(* Logix 5000 project; controller Sucrose_Main Emulate 5570 rev 20.12; software revision 20.01; part 28 of 30 *)
(* tags used below, declared in another part *)
   AI_E23_0 : REAL[8];   // Analog Input EN2T_FLX 192.168.1.23
   AI_E23_1 : REAL[8];   // Analog Input EN2T_FLX 192.168.1.23
   Alarm_ACK_Master_Timer : TIMER;
   DI_E23_3 : ALIAS FOR FLX_E23:3:I;   // Discrete Input EN2T_FLX 192.168.1.23
   DO_E24_3 : ALIAS FOR FLX_E24:3:O;   // Discrete Output EN2T_FLX 192.168.1.24
   FV230102_AOI : QSI_Flow_Valve;   // FV-23-01-02 SUCROSE TANK #1 INLET/SPRAYBALL VALVE
   FV230104_AOI : QSI_Flow_Valve;   // FV-23-01-04-O SUCROSE RETURN TO SUCROSE TANK #1 VALVE OPEN
   FV230204_AOI : QSI_Flow_Valve;   // FV-23-02-04-O SUCROSE RETURN TO SUCROSE TANK #2 VALVE OPEN
   FV230222_AOI : QSI_Flow_Valve;   // FV-23-02-22-O SUCROSE TANK #2 TO TRANSFER PUMP #2 MIX PROOF VALVE OPEN
   FV230304_AOI : QSI_Flow_Valve;   // FV-23-03-04-O SUCROSE RETURN TO SUCROSE TANK #3 VALVE OPEN
   FV230411_AOI : QSI_Flow_Valve;   // FV-23-04-11-O SUCROSE TANK #1 TO TRANSFER PUMP #1 MIX PROOF VALVE OPEN
   FV230412_AOI : QSI_Flow_Valve;   // FV-23-04-12-O SUCROSE TANK #2 TO TRANSFER PUMP #1 MIX PROOF VALVE OPEN
   FV230413_AOI : QSI_Flow_Valve;   // FV-23-04-13-O SUCROSE TANK #3 TO TRANSFER PUMP #1 MIX PROOF VALVE OPEN
   FV230421_AOI : QSI_Flow_Valve;   // FV-23-04-21-O SUCROSE TANK #1 TO TRANSFER PUMP #2 MIX PROOF VALVE OPEN
   FV230423_AOI : QSI_Flow_Valve;   // FV-23-04-23-O SUCROSE TANK #3 TO TRANSFER PUMP #2 MIX PROOF VALVE OPEN
   FV751101_AOI : QSI_Flow_Valve;   // FV-75-11-01 SUCROSE TANK #1 BLANKETING STEAM TRAP ISOLATION VALVE
   FV931101_AOI : QSI_Flow_Valve;   // FV-93-11-01 STERILE AIR FLT-93-11-01 SHUT OFF VALVE
   ONESHOTBITS : INT[10];
   Rung_Comment : BOOL;
   Sucrose_MM_Enable : BOOL;
   SucroseCIP_RINGMAIN_REMOTE : CIP_REMOTE;
   SucroseCIP_TK230101_REMOTE : CIP_REMOTE;
   SucroseCIP_TK230201_REMOTE : CIP_REMOTE;
   SucroseCIP_TK230301_REMOTE : CIP_REMOTE;
   SucroseDischarge : Area_Program;
   SucroseFiltration : Area_Program;
   SucroseTanks : Area_Program;
   TK_23_01_01_HEALOUT_TIME_REMAINING : DINT;
   TK_23_01_01_LOW_LEVEL : DINT;
   TK_23_01_01_NO_PRESS_ALARM : BOOL;
   TK_23_01_01_NO_TEMP_ALARM : BOOL;
   TK_23_02_01_HEALOUT_TIME_REMAINING : DINT;
   TK_23_02_01_LOW_LEVEL : DINT;
   TK_23_02_01_NO_PRESS_ALARM : BOOL;
   TK_23_02_01_NO_TEMP_ALARM : BOOL;
   TK_23_03_01_HEALOUT_TIME_REMAINING : DINT;
   TK_23_03_01_LOW_LEVEL : DINT;
   TK_23_03_01_NO_PRESS_ALARM : BOOL;
   TK_23_03_01_NO_TEMP_ALARM : BOOL;
(* TanksArea_AutoLogic, continued *)

ROUTINE Control_Logic   (* ladder *)
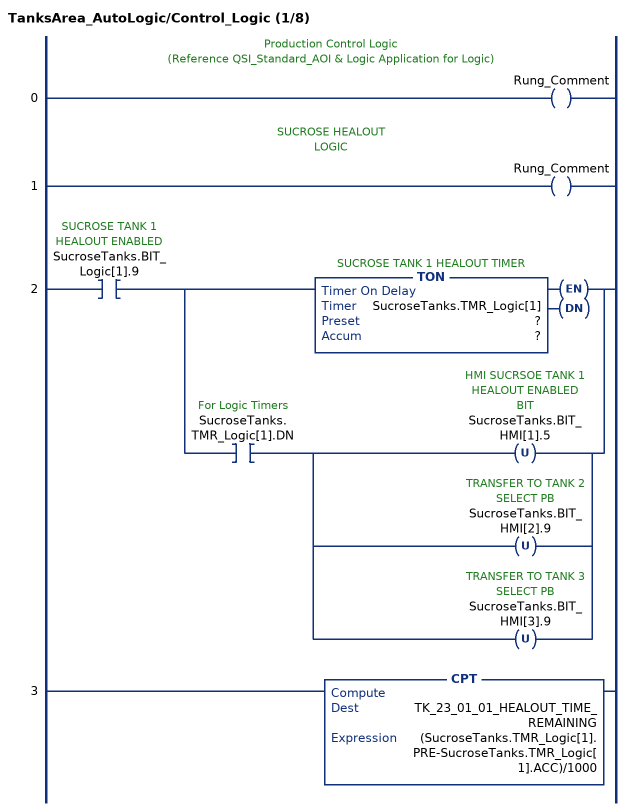
   // Production Control Logic
   // (Reference QSI_Standard_AOI & Logic Application for Logic)
   0: OTE(Rung_Comment);
   // SUCROSE HEALOUT
   // LOGIC
   1: OTE(Rung_Comment);
   2: XIC(SucroseTanks.BIT_Logic[1].9)[TON(SucroseTanks.TMR_Logic[1],?,?) ,XIC(SucroseTanks.TMR_Logic[1].DN) [OTU(SucroseTanks.BIT_HMI[1].5) ,OTU(SucroseTanks.BIT_HMI[2].9) ,OTU(SucroseTanks.BIT_HMI[3].9) ] ];
   3: CPT(TK_23_01_01_HEALOUT_TIME_REMAINING,(SucroseTanks.TMR_Logic[1].PRE-SucroseTanks.TMR_Logic[1].ACC)/1000);
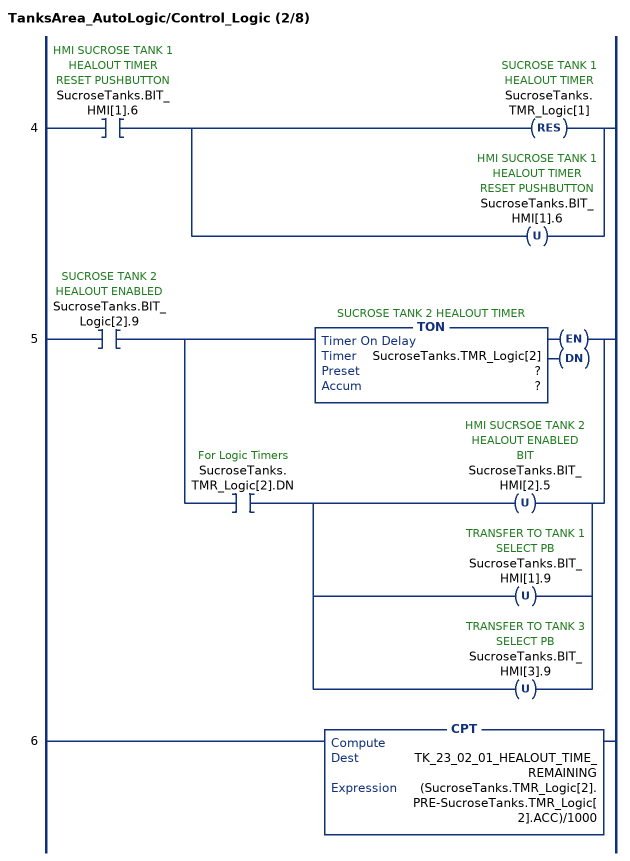
   4: XIC(SucroseTanks.BIT_HMI[1].6)[RES(SucroseTanks.TMR_Logic[1]) ,OTU(SucroseTanks.BIT_HMI[1].6) ];
   5: XIC(SucroseTanks.BIT_Logic[2].9)[TON(SucroseTanks.TMR_Logic[2],?,?) ,XIC(SucroseTanks.TMR_Logic[2].DN) [OTU(SucroseTanks.BIT_HMI[2].5) ,OTU(SucroseTanks.BIT_HMI[1].9) ,OTU(SucroseTanks.BIT_HMI[3].9) ] ];
   6: CPT(TK_23_02_01_HEALOUT_TIME_REMAINING,(SucroseTanks.TMR_Logic[2].PRE-SucroseTanks.TMR_Logic[2].ACC)/1000);
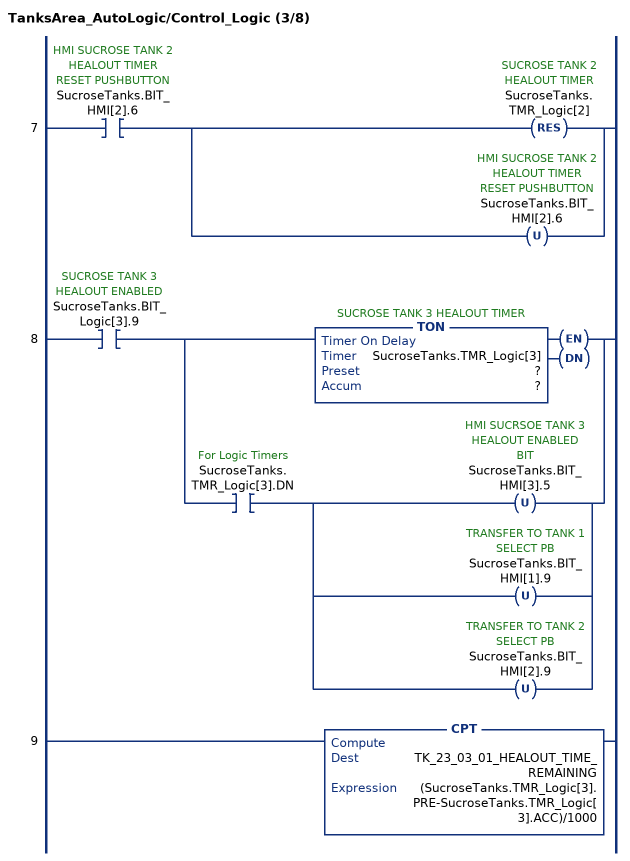
   7: XIC(SucroseTanks.BIT_HMI[2].6)[RES(SucroseTanks.TMR_Logic[2]) ,OTU(SucroseTanks.BIT_HMI[2].6) ];
   8: XIC(SucroseTanks.BIT_Logic[3].9)[TON(SucroseTanks.TMR_Logic[3],?,?) ,XIC(SucroseTanks.TMR_Logic[3].DN) [OTU(SucroseTanks.BIT_HMI[3].5) ,OTU(SucroseTanks.BIT_HMI[1].9) ,OTU(SucroseTanks.BIT_HMI[2].9) ] ];
   9: CPT(TK_23_03_01_HEALOUT_TIME_REMAINING,(SucroseTanks.TMR_Logic[3].PRE-SucroseTanks.TMR_Logic[3].ACC)/1000);
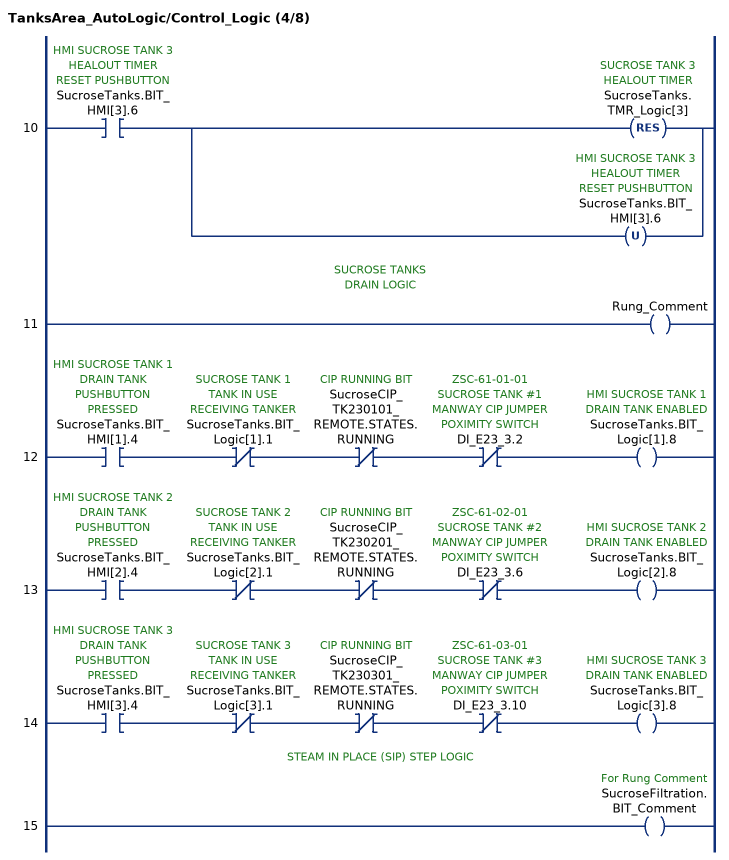
   10: XIC(SucroseTanks.BIT_HMI[3].6)[RES(SucroseTanks.TMR_Logic[3]) ,OTU(SucroseTanks.BIT_HMI[3].6) ];
   // SUCROSE TANKS
   // DRAIN LOGIC
   11: OTE(Rung_Comment);
   12: XIC(SucroseTanks.BIT_HMI[1].4)XIO(SucroseTanks.BIT_Logic[1].1)XIO(SucroseCIP_TK230101_REMOTE.STATES.RUNNING)XIO(DI_E23_3.2)OTE(SucroseTanks.BIT_Logic[1].8);
   13: XIC(SucroseTanks.BIT_HMI[2].4)XIO(SucroseTanks.BIT_Logic[2].1)XIO(SucroseCIP_TK230201_REMOTE.STATES.RUNNING)XIO(DI_E23_3.6)OTE(SucroseTanks.BIT_Logic[2].8);
   14: XIC(SucroseTanks.BIT_HMI[3].4)XIO(SucroseTanks.BIT_Logic[3].1)XIO(SucroseCIP_TK230301_REMOTE.STATES.RUNNING)XIO(DI_E23_3.10)OTE(SucroseTanks.BIT_Logic[3].8);
   // STEAM IN PLACE (SIP) STEP LOGIC
   15: OTE(SucroseFiltration.BIT_Comment);
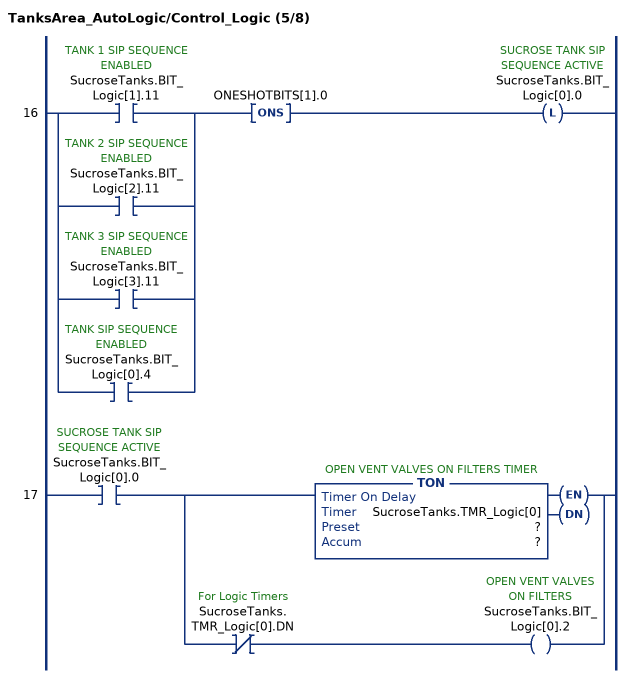
   16: [XIC(SucroseTanks.BIT_Logic[1].11) ,XIC(SucroseTanks.BIT_Logic[2].11) ,XIC(SucroseTanks.BIT_Logic[3].11) ,XIC(SucroseTanks.BIT_Logic[0].4) ]ONS(ONESHOTBITS[1].0)OTL(SucroseTanks.BIT_Logic[0].0);
   17: XIC(SucroseTanks.BIT_Logic[0].0)[TON(SucroseTanks.TMR_Logic[0],?,?) ,XIO(SucroseTanks.TMR_Logic[0].DN) OTE(SucroseTanks.BIT_Logic[0].2) ];
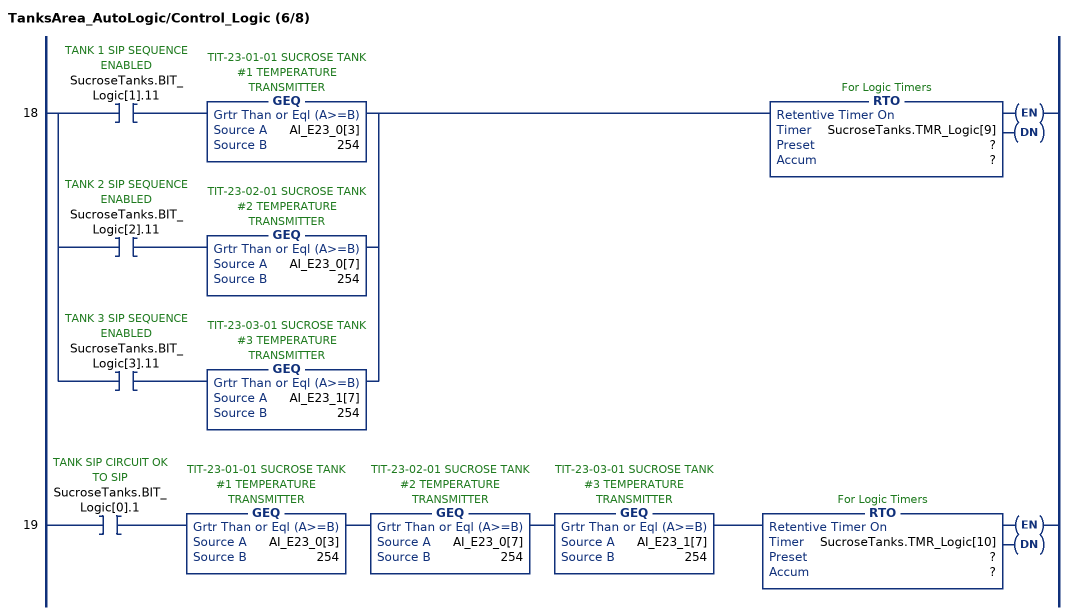
   18: [XIC(SucroseTanks.BIT_Logic[1].11) GEQ(AI_E23_0[3],254) ,XIC(SucroseTanks.BIT_Logic[2].11) GEQ(AI_E23_0[7],254) ,XIC(SucroseTanks.BIT_Logic[3].11) GEQ(AI_E23_1[7],254) ]RTO(SucroseTanks.TMR_Logic[9],?,?);
   19: XIC(SucroseTanks.BIT_Logic[0].1)GEQ(AI_E23_0[3],254)GEQ(AI_E23_0[7],254)GEQ(AI_E23_1[7],254)RTO(SucroseTanks.TMR_Logic[10],?,?);
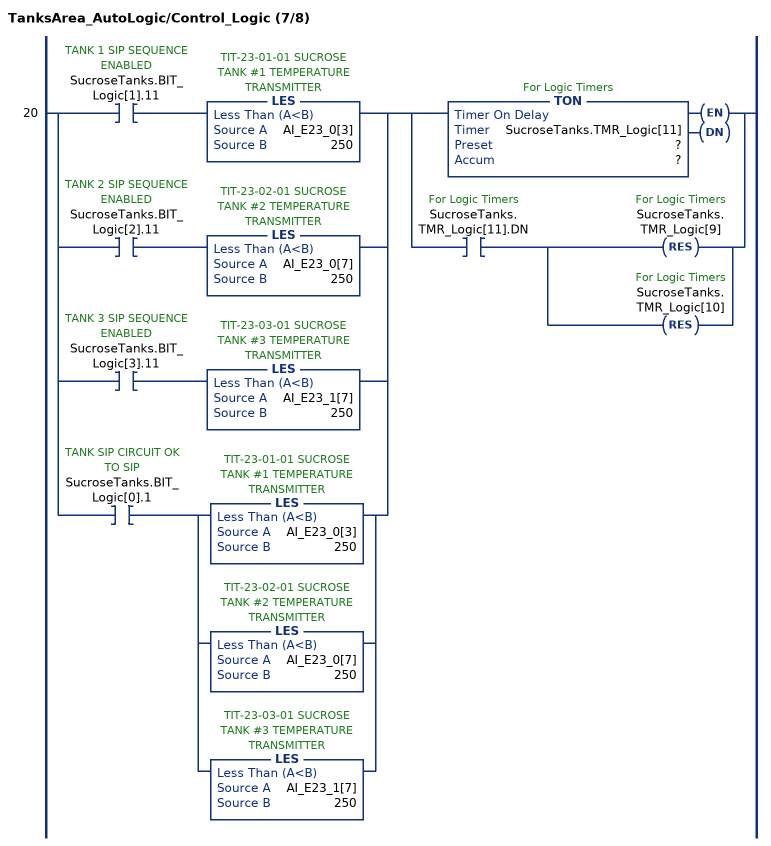
   20: [XIC(SucroseTanks.BIT_Logic[1].11) LES(AI_E23_0[3],250) ,XIC(SucroseTanks.BIT_Logic[2].11) LES(AI_E23_0[7],250) ,XIC(SucroseTanks.BIT_Logic[3].11) LES(AI_E23_1[7],250) ,XIC(SucroseTanks.BIT_Logic[0].1) [LES(AI_E23_0[3],250) ,LES(AI_E23_0[7],250) ,LES(AI_E23_1[7],250) ] ][TON(SucroseTanks.TMR_Logic[11],?,?) ,XIC(SucroseTanks.TMR_Logic[11].DN) [RES(SucroseTanks.TMR_Logic[9]) ,RES(SucroseTanks.TMR_Logic[10]) ] ];
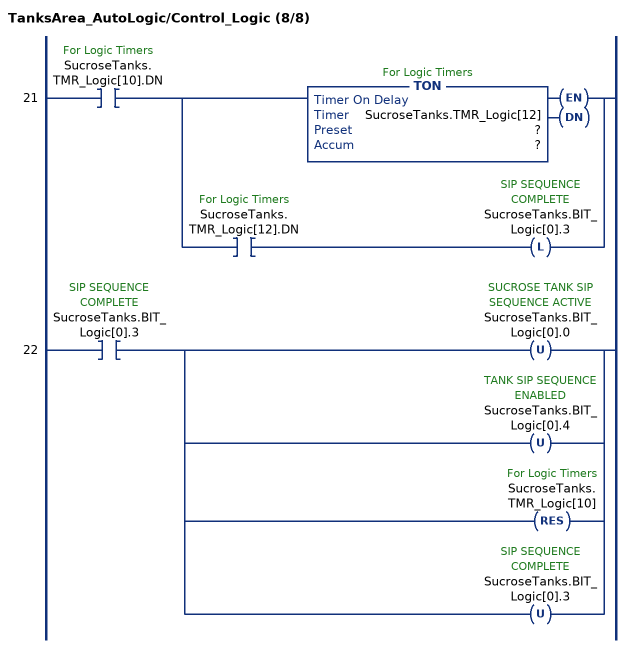
   21: XIC(SucroseTanks.TMR_Logic[10].DN)[TON(SucroseTanks.TMR_Logic[12],?,?) ,XIC(SucroseTanks.TMR_Logic[12].DN) OTL(SucroseTanks.BIT_Logic[0].3) ];
   22: XIC(SucroseTanks.BIT_Logic[0].3)[OTU(SucroseTanks.BIT_Logic[0].0) ,OTU(SucroseTanks.BIT_Logic[0].4) ,RES(SucroseTanks.TMR_Logic[10]) ,OTU(SucroseTanks.BIT_Logic[0].3) ];
END_ROUTINE

ROUTINE Enable_Logic   (* ladder *)
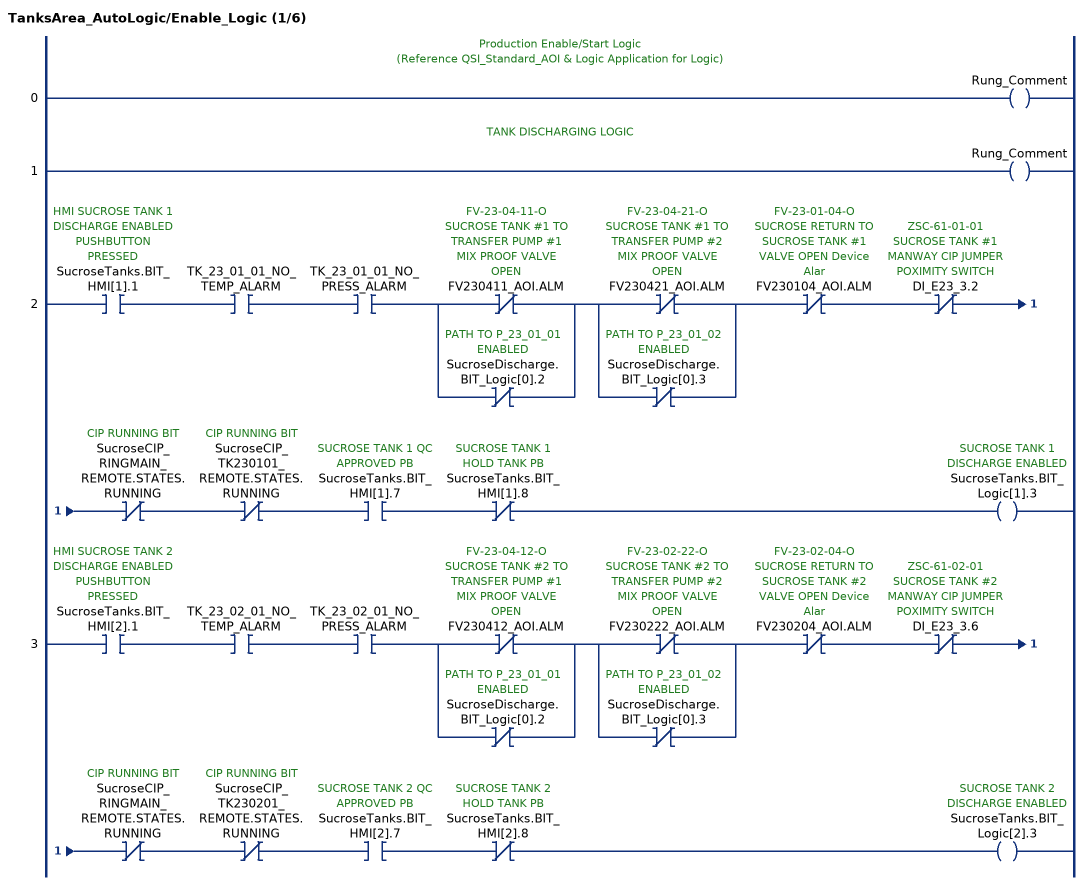
   // Production Enable/Start Logic
   // (Reference QSI_Standard_AOI & Logic Application for Logic)
   0: OTE(Rung_Comment);
   // TANK DISCHARGING LOGIC
   1: OTE(Rung_Comment);
   2: XIC(SucroseTanks.BIT_HMI[1].1)XIC(TK_23_01_01_NO_TEMP_ALARM)XIC(TK_23_01_01_NO_PRESS_ALARM)[XIO(FV230411_AOI.ALM) ,XIO(SucroseDischarge.BIT_Logic[0].2) ][XIO(FV230421_AOI.ALM) ,XIO(SucroseDischarge.BIT_Logic[0].3) ]XIO(FV230104_AOI.ALM)XIO(DI_E23_3.2)XIO(SucroseCIP_RINGMAIN_REMOTE.STATES.RUNNING)XIO(SucroseCIP_TK230101_REMOTE.STATES.RUNNING)XIC(SucroseTanks.BIT_HMI[1].7)XIO(SucroseTanks.BIT_HMI[1].8)OTE(SucroseTanks.BIT_Logic[1].3);
   3: XIC(SucroseTanks.BIT_HMI[2].1)XIC(TK_23_02_01_NO_TEMP_ALARM)XIC(TK_23_02_01_NO_PRESS_ALARM)[XIO(FV230412_AOI.ALM) ,XIO(SucroseDischarge.BIT_Logic[0].2) ][XIO(FV230222_AOI.ALM) ,XIO(SucroseDischarge.BIT_Logic[0].3) ]XIO(FV230204_AOI.ALM)XIO(DI_E23_3.6)XIO(SucroseCIP_RINGMAIN_REMOTE.STATES.RUNNING)XIO(SucroseCIP_TK230201_REMOTE.STATES.RUNNING)XIC(SucroseTanks.BIT_HMI[2].7)XIO(SucroseTanks.BIT_HMI[2].8)OTE(SucroseTanks.BIT_Logic[2].3);
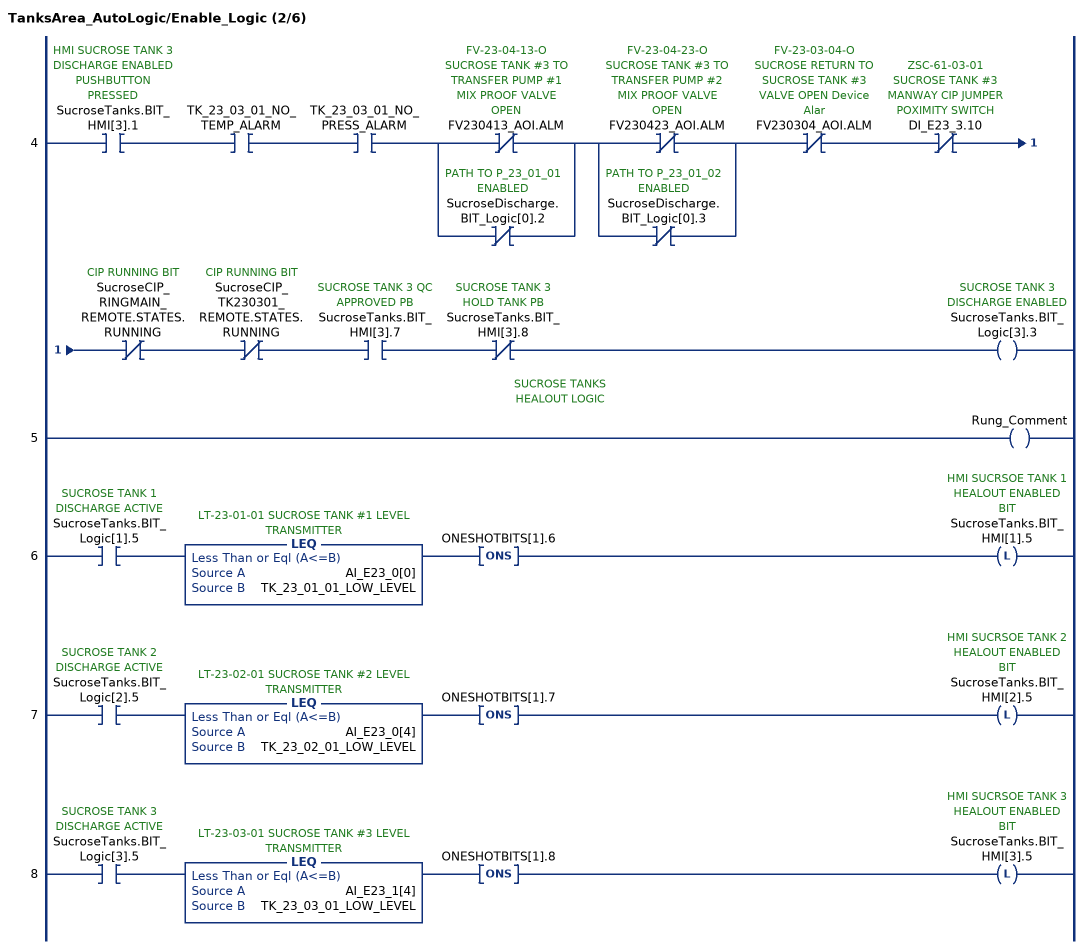
   4: XIC(SucroseTanks.BIT_HMI[3].1)XIC(TK_23_03_01_NO_TEMP_ALARM)XIC(TK_23_03_01_NO_PRESS_ALARM)[XIO(FV230413_AOI.ALM) ,XIO(SucroseDischarge.BIT_Logic[0].2) ][XIO(FV230423_AOI.ALM) ,XIO(SucroseDischarge.BIT_Logic[0].3) ]XIO(FV230304_AOI.ALM)XIO(DI_E23_3.10)XIO(SucroseCIP_RINGMAIN_REMOTE.STATES.RUNNING)XIO(SucroseCIP_TK230301_REMOTE.STATES.RUNNING)XIC(SucroseTanks.BIT_HMI[3].7)XIO(SucroseTanks.BIT_HMI[3].8)OTE(SucroseTanks.BIT_Logic[3].3);
   // SUCROSE TANKS
   // HEALOUT LOGIC
   5: OTE(Rung_Comment);
   6: XIC(SucroseTanks.BIT_Logic[1].5)LEQ(AI_E23_0[0],TK_23_01_01_LOW_LEVEL)ONS(ONESHOTBITS[1].6)OTL(SucroseTanks.BIT_HMI[1].5);
   7: XIC(SucroseTanks.BIT_Logic[2].5)LEQ(AI_E23_0[4],TK_23_02_01_LOW_LEVEL)ONS(ONESHOTBITS[1].7)OTL(SucroseTanks.BIT_HMI[2].5);
   8: XIC(SucroseTanks.BIT_Logic[3].5)LEQ(AI_E23_1[4],TK_23_03_01_LOW_LEVEL)ONS(ONESHOTBITS[1].8)OTL(SucroseTanks.BIT_HMI[3].5);
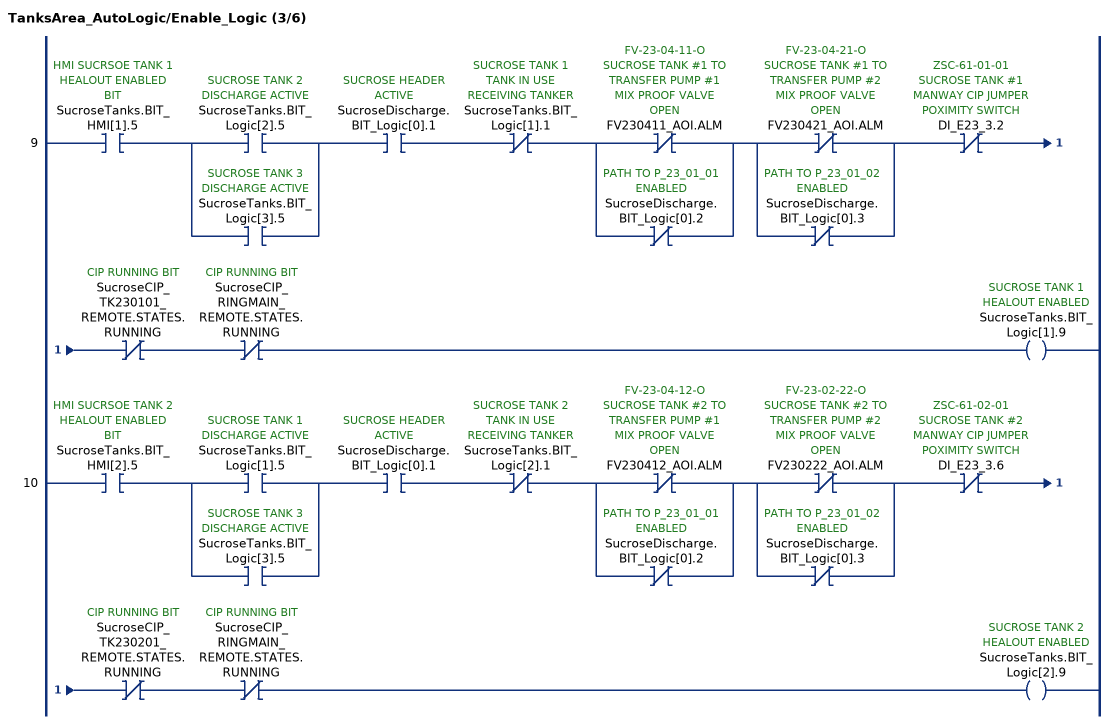
   9: XIC(SucroseTanks.BIT_HMI[1].5)[XIC(SucroseTanks.BIT_Logic[2].5) ,XIC(SucroseTanks.BIT_Logic[3].5) ]XIC(SucroseDischarge.BIT_Logic[0].1)XIO(SucroseTanks.BIT_Logic[1].1)[XIO(FV230411_AOI.ALM) ,XIO(SucroseDischarge.BIT_Logic[0].2) ][XIO(FV230421_AOI.ALM) ,XIO(SucroseDischarge.BIT_Logic[0].3) ]XIO(DI_E23_3.2)XIO(SucroseCIP_TK230101_REMOTE.STATES.RUNNING)XIO(SucroseCIP_RINGMAIN_REMOTE.STATES.RUNNING)OTE(SucroseTanks.BIT_Logic[1].9);
   10: XIC(SucroseTanks.BIT_HMI[2].5)[XIC(SucroseTanks.BIT_Logic[1].5) ,XIC(SucroseTanks.BIT_Logic[3].5) ]XIC(SucroseDischarge.BIT_Logic[0].1)XIO(SucroseTanks.BIT_Logic[2].1)[XIO(FV230412_AOI.ALM) ,XIO(SucroseDischarge.BIT_Logic[0].2) ][XIO(FV230222_AOI.ALM) ,XIO(SucroseDischarge.BIT_Logic[0].3) ]XIO(DI_E23_3.6)XIO(SucroseCIP_TK230201_REMOTE.STATES.RUNNING)XIO(SucroseCIP_RINGMAIN_REMOTE.STATES.RUNNING)OTE(SucroseTanks.BIT_Logic[2].9);
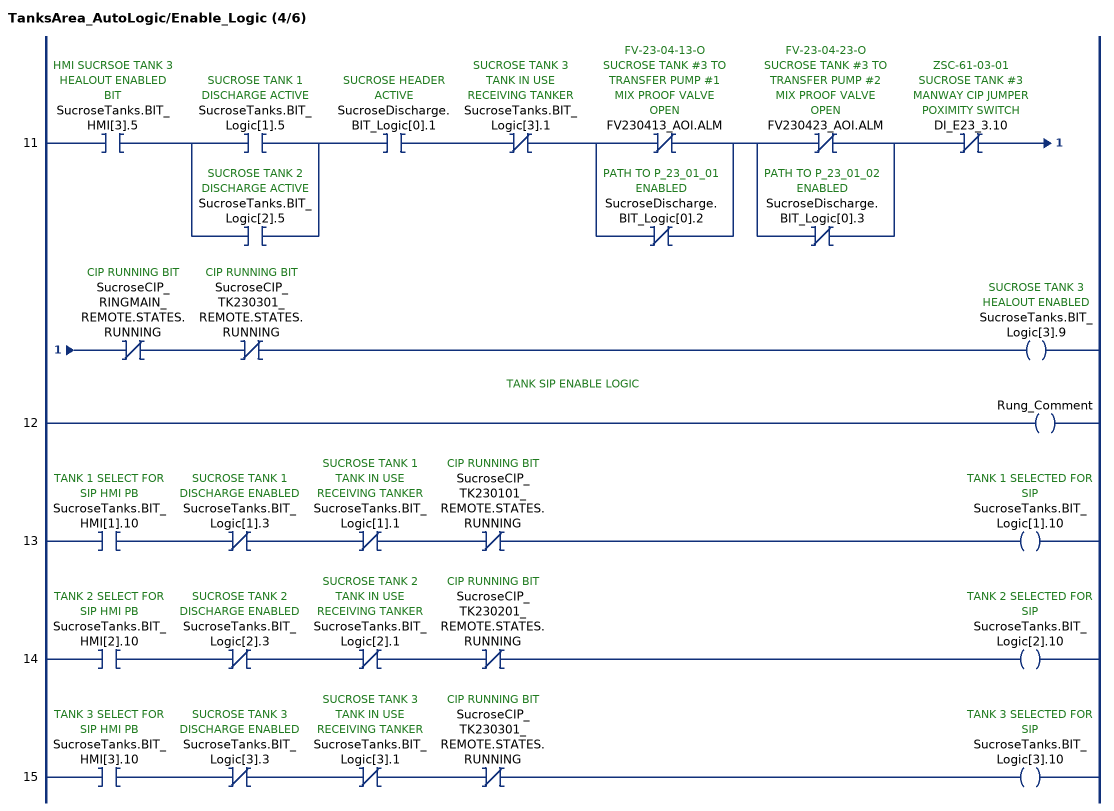
   11: XIC(SucroseTanks.BIT_HMI[3].5)[XIC(SucroseTanks.BIT_Logic[1].5) ,XIC(SucroseTanks.BIT_Logic[2].5) ]XIC(SucroseDischarge.BIT_Logic[0].1)XIO(SucroseTanks.BIT_Logic[3].1)[XIO(FV230413_AOI.ALM) ,XIO(SucroseDischarge.BIT_Logic[0].2) ][XIO(FV230423_AOI.ALM) ,XIO(SucroseDischarge.BIT_Logic[0].3) ]XIO(DI_E23_3.10)XIO(SucroseCIP_RINGMAIN_REMOTE.STATES.RUNNING)XIO(SucroseCIP_TK230301_REMOTE.STATES.RUNNING)OTE(SucroseTanks.BIT_Logic[3].9);
   // TANK SIP ENABLE LOGIC
   12: OTE(Rung_Comment);
   13: XIC(SucroseTanks.BIT_HMI[1].10)XIO(SucroseTanks.BIT_Logic[1].3)XIO(SucroseTanks.BIT_Logic[1].1)XIO(SucroseCIP_TK230101_REMOTE.STATES.RUNNING)OTE(SucroseTanks.BIT_Logic[1].10);
   14: XIC(SucroseTanks.BIT_HMI[2].10)XIO(SucroseTanks.BIT_Logic[2].3)XIO(SucroseTanks.BIT_Logic[2].1)XIO(SucroseCIP_TK230201_REMOTE.STATES.RUNNING)OTE(SucroseTanks.BIT_Logic[2].10);
   15: XIC(SucroseTanks.BIT_HMI[3].10)XIO(SucroseTanks.BIT_Logic[3].3)XIO(SucroseTanks.BIT_Logic[3].1)XIO(SucroseCIP_TK230301_REMOTE.STATES.RUNNING)OTE(SucroseTanks.BIT_Logic[3].10);
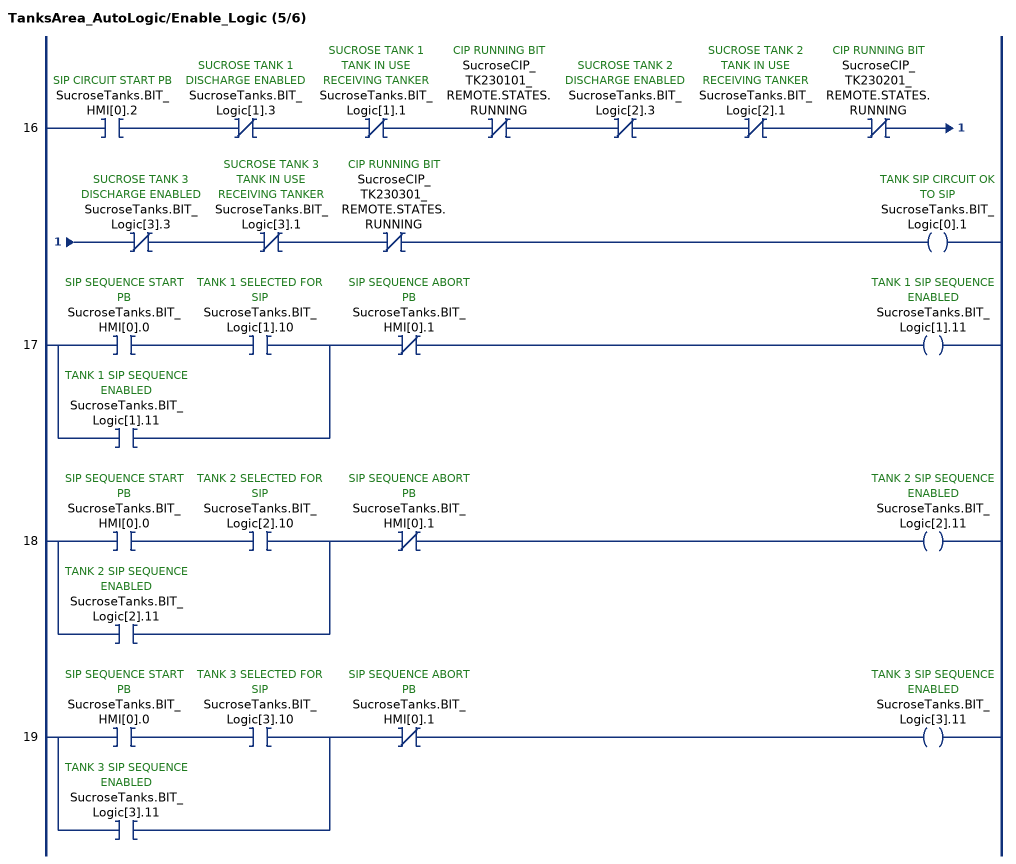
   16: XIC(SucroseTanks.BIT_HMI[0].2)XIO(SucroseTanks.BIT_Logic[1].3)XIO(SucroseTanks.BIT_Logic[1].1)XIO(SucroseCIP_TK230101_REMOTE.STATES.RUNNING)XIO(SucroseTanks.BIT_Logic[2].3)XIO(SucroseTanks.BIT_Logic[2].1)XIO(SucroseCIP_TK230201_REMOTE.STATES.RUNNING)XIO(SucroseTanks.BIT_Logic[3].3)XIO(SucroseTanks.BIT_Logic[3].1)XIO(SucroseCIP_TK230301_REMOTE.STATES.RUNNING)OTE(SucroseTanks.BIT_Logic[0].1);
   17: [XIC(SucroseTanks.BIT_HMI[0].0) XIC(SucroseTanks.BIT_Logic[1].10) ,XIC(SucroseTanks.BIT_Logic[1].11) ]XIO(SucroseTanks.BIT_HMI[0].1)OTE(SucroseTanks.BIT_Logic[1].11);
   18: [XIC(SucroseTanks.BIT_HMI[0].0) XIC(SucroseTanks.BIT_Logic[2].10) ,XIC(SucroseTanks.BIT_Logic[2].11) ]XIO(SucroseTanks.BIT_HMI[0].1)OTE(SucroseTanks.BIT_Logic[2].11);
   19: [XIC(SucroseTanks.BIT_HMI[0].0) XIC(SucroseTanks.BIT_Logic[3].10) ,XIC(SucroseTanks.BIT_Logic[3].11) ]XIO(SucroseTanks.BIT_HMI[0].1)OTE(SucroseTanks.BIT_Logic[3].11);
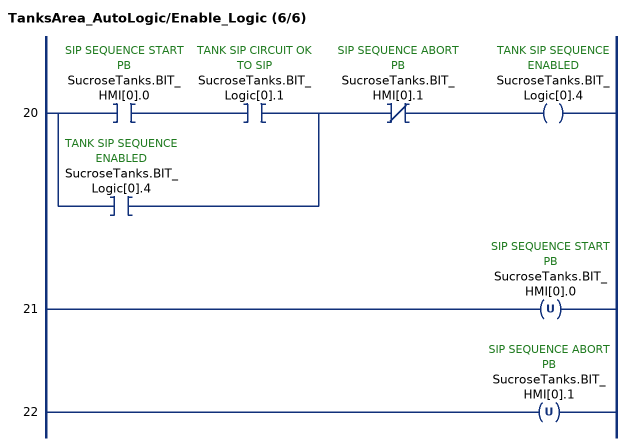
   20: [XIC(SucroseTanks.BIT_HMI[0].0) XIC(SucroseTanks.BIT_Logic[0].1) ,XIC(SucroseTanks.BIT_Logic[0].4) ]XIO(SucroseTanks.BIT_HMI[0].1)OTE(SucroseTanks.BIT_Logic[0].4);
   21: OTU(SucroseTanks.BIT_HMI[0].0);
   22: OTU(SucroseTanks.BIT_HMI[0].1);
END_ROUTINE

ROUTINE MainRoutine   (* ladder *)
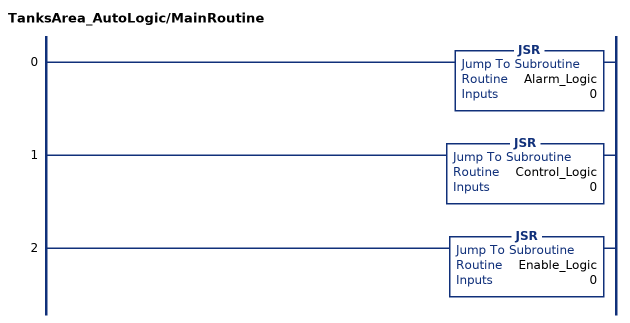
   0: JSR(Alarm_Logic,0);
   1: JSR(Control_Logic,0);
   2: JSR(Enable_Logic,0);
END_ROUTINE
END_PROGRAM

PROGRAM TanksArea_EN2T_IO_Discrete_DO_E24_3   (* main routine MainRoutine *)

ROUTINE _00_FV230102   (* ladder *)
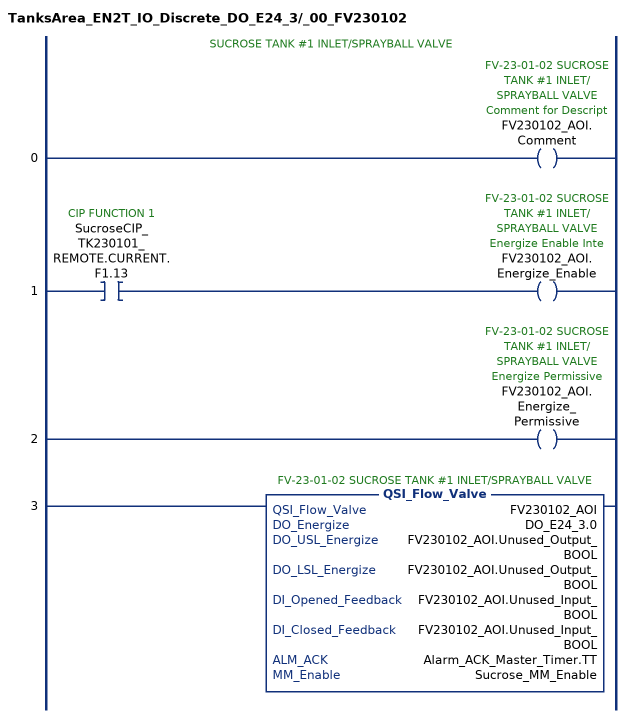
   // SUCROSE TANK #1 INLET/SPRAYBALL VALVE
   0: OTE(FV230102_AOI.Comment);
   1: XIC(SucroseCIP_TK230101_REMOTE.CURRENT.F1.13)OTE(FV230102_AOI.Energize_Enable);
   2: OTE(FV230102_AOI.Energize_Permissive);
   3: QSI_Flow_Valve(FV230102_AOI,DO_E24_3.0,FV230102_AOI.Unused_Output_BOOL,FV230102_AOI.Unused_Output_BOOL,FV230102_AOI.Unused_Input_BOOL,FV230102_AOI.Unused_Input_BOOL,Alarm_ACK_Master_Timer.TT,Sucrose_MM_Enable);
END_ROUTINE

ROUTINE _02_FV751101   (* ladder *)
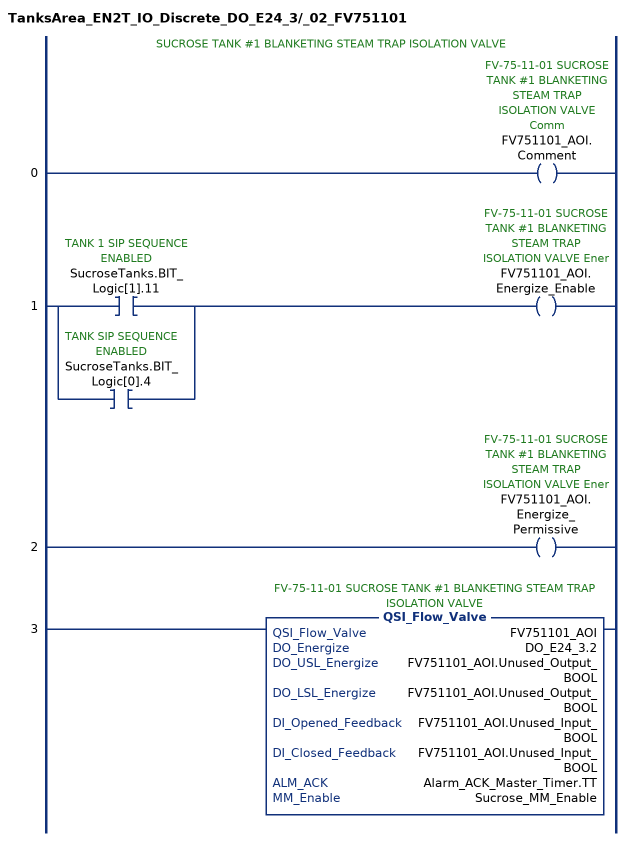
   // SUCROSE TANK #1 BLANKETING STEAM TRAP ISOLATION VALVE
   0: OTE(FV751101_AOI.Comment);
   1: [XIC(SucroseTanks.BIT_Logic[1].11) ,XIC(SucroseTanks.BIT_Logic[0].4) ]OTE(FV751101_AOI.Energize_Enable);
   2: OTE(FV751101_AOI.Energize_Permissive);
   3: QSI_Flow_Valve(FV751101_AOI,DO_E24_3.2,FV751101_AOI.Unused_Output_BOOL,FV751101_AOI.Unused_Output_BOOL,FV751101_AOI.Unused_Input_BOOL,FV751101_AOI.Unused_Input_BOOL,Alarm_ACK_Master_Timer.TT,Sucrose_MM_Enable);
END_ROUTINE

ROUTINE _03_FV931101   (* ladder *)
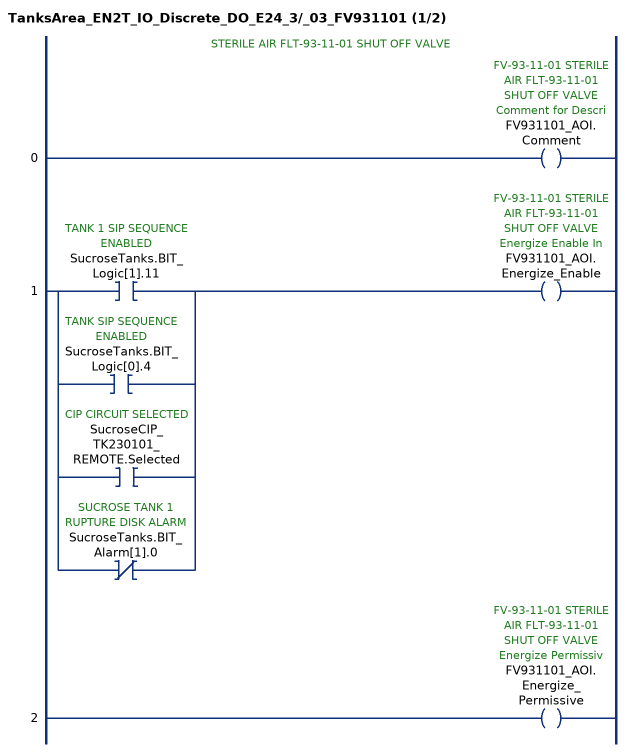
   // STERILE AIR FLT-93-11-01 SHUT OFF VALVE
   0: OTE(FV931101_AOI.Comment);
   1: [XIC(SucroseTanks.BIT_Logic[1].11) ,XIC(SucroseTanks.BIT_Logic[0].4) ,XIC(SucroseCIP_TK230101_REMOTE.Selected) ,XIO(SucroseTanks.BIT_Alarm[1].0) ]OTE(FV931101_AOI.Energize_Enable);
   2: OTE(FV931101_AOI.Energize_Permissive);
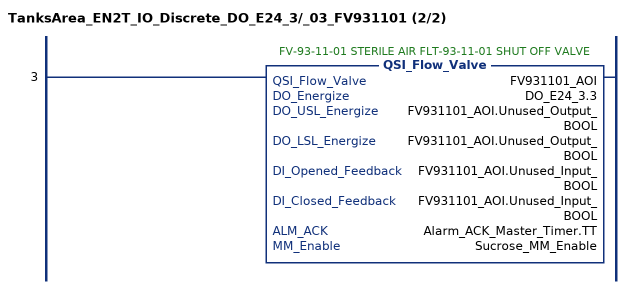
   3: QSI_Flow_Valve(FV931101_AOI,DO_E24_3.3,FV931101_AOI.Unused_Output_BOOL,FV931101_AOI.Unused_Output_BOOL,FV931101_AOI.Unused_Input_BOOL,FV931101_AOI.Unused_Input_BOOL,Alarm_ACK_Master_Timer.TT,Sucrose_MM_Enable);
END_ROUTINE
